TYPE ST_HMI_TRAFFIC_LIGHT_OUT :
STRUCT
	bLedGN	: BOOL;
	bLedGE	: BOOL;
	bLedRT	: BOOL;
	bLedBL	: BOOL;
END_STRUCT
END_TYPE

(* stored: Version 1.1.0.1
   DUT ST_HMI_TRAFFIC_LIGHT_OUT: Id {ab4a16ea-cce9-489b-ac4b-9a8dc188adcc} *)
